(* PLC project PLC, Beckhoff Automation GmbH TwinCAT PLC Control 3.5.13.21 *)
(* stored: creationDateTime 2023-01-03T15:24:25.9685047, modificationDateTime 2023-01-03T15:24:25.9685047 *)

PROGRAM AutoGenerated
  VAR
    Step : INT;
    StepReadEtherCATDiagnostics : INT;
    TonReadDiagnostics : TON;
    sError : STRING;
    FB_EcCoESdoWrite1 : FB_EcCoESdoWrite;
    CoEWriteBuffer : DWORD;
    FB_EcMasterFrameStatisticClearTxRxErr : FB_EcMasterFrameStatisticClearTxRxErr;
    FB_EcGetAllSlavePresentStateChanges : FB_EcGetAllSlavePresentStateChanges;
    fbGetAllSlaveStates : FB_EcGetAllSlaveStates;
    fbEcGetConfSlaves : FB_EcGetConfSlaves;
    fbEcGetAllSlaveCrcErrors : FB_EcGetAllSlaveCrcErrors;
    stSlaveStates : ARRAY[0..EtherDeviceCount] OF ST_EcSlaveState;
    stArrEcConfSlaveInfo : ARRAY[0..EtherDeviceCount] OF ST_EcSlaveConfigData;
    dwArrSlaveCrcCount : ARRAY[0..EtherDeviceCount] OF DWORD;
    dwArrSlaveChangeCount : ARRAY[0..EtherDeviceCount] OF DWORD;
    dwArrSlaveChangeCountHistory : ARRAY[0..EtherDeviceCount] OF DWORD;
    bExecuteFB_GetAdaptersInfo : BOOL := TRUE;  (* /////// Set IP address////////////// *)
    NICCount : INT := 2;
    NicIndex : INT := 1;
    FB_GetAdaptersInfo : FB_GetAdaptersInfo;
    fbDiagRegister : FB_IPCDiag_Register := (sNetId := '');
    fbWriteNicInfo : FB_IPCDiag_WriteParameter;
    iPrevState : INT;
    iState : INT;
    _usiModuleIndex : USINT;
    _sIPAddress : STRING;
    _sIPSubNetMask : STRING;
    _sIPGateway : STRING;
    _xDHCP : BOOL;
    rtExecuteTrig : R_TRIG;
    xBusy : BOOL;
    xError : BOOL;
    hrErrorCode : HRESULT;
    xExecute : BOOL;
    usiModuleIndex : USINT;
    sIPAddress : STRING;
    sIPSubnetMask : STRING;
    sIPGateway : STRING;
    xDHCP : BOOL;
    sCurrentNicName : STRING;
    FB_EcMasterFrameStatisticClearFrames : FB_EcMasterFrameStatisticClearFrames;
    StepCoERead : UDINT;  (* //// End IP address // Start CoE read *)
    CoEReadPos : INT;
    CoEReadbytePos : INT;
    CoEReadintPos : INT;
    CoEReaduintPos : INT;
    CoEReadudintPos : INT;
    CoEReadboolPos : INT;
    fbCoERead : FB_EcCoESdoReadEx;
    CoEReadcbBufLen : ARRAY[1..CoEReadTotalCount] OF UDINT;  (* CoEReadIndex : ARRAY[1..50] OF WORD; CoEReadSubIndex : ARRAY[1..50] OF BYTE; CoEReadSlaveAddr : ARRAY[1..50] OF UINT; *)
    CoEReadData : ARRAY[1..CoEReadTotalCount] OF POINTER TO BYTE;
    CoEReadErrorCounter : UDINT;
    CoEReadErrorIndex : UDINT;
    CoEReadTonUpdateRate : TON;
    i : UDINT;
  END_VAR

            EtherCAT_Diagnostics();

SetIpAddress();
stArrEcConfSlaveInfo[1].sName;
stArrEcConfSlaveInfo[1].sType;
stArrEcConfSlaveInfo[1].nAddr;

CASE StepCoERead OF //Cyclicly read CoE data to send back to rockwell controller.
	0: //This step is important because it sets all the pointer values. 
	
		CoEReadintPos:=0;
		//Not implimented yet.
		CoEReadPos:=1;
		StepCoERead:=StepCoERead+10;
		//Update Pointers
		FOR i:=1 TO  CoEReadTotalCount BY 1 DO
			IF CoEReadDataType[i] = 'INT' THEN
				CoEReadintPos:=CoEReadintPos+1;
				CoEReadData[i]:=ADR(CoEReadInt[CoEReadintPos]);
				CoEReadcbBufLen[i]:=SIZEOF(CoEReadInt[CoEReadintPos]);
			ELSIF CoEReadDataType[i] = 'BYTE' THEN
				CoEReadbytePos:=CoEReadbytePos+1;
				CoEReadData[i]:=ADR(CoEReadByte[CoEReadbytePos]);
				CoEReadcbBufLen[i]:=SIZEOF(CoEReadByte[CoEReadbytePos]);
			ELSIF CoEReadDataType[i] = 'UINT' THEN
				CoEReaduintPos:=CoEReaduintPos+1;
				CoEReadData[i]:=ADR(CoEReadUint[CoEReaduintPos]);
				CoEReadcbBufLen[i]:=SIZEOF(CoEReadUint[CoEReaduintPos]);
			ELSIF CoEReadDataType[i] = 'UDINT' THEN
				CoEReadudintPos:=CoEReadudintPos+1;
				CoEReadData[i]:=ADR(CoEReadUdint[CoEReadudintPos]);
				CoEReadcbBufLen[i]:=SIZEOF(CoEReadUdint[CoEReadudintPos]);
			ELSIF CoEReadDataType[i] = 'BOOL' THEN
				CoEReadboolPos:=CoEReadboolPos+1;
				CoEReadData[i]:=ADR(CoEReadBool[CoEReadboolPos]);
				CoEReadcbBufLen[i]:=SIZEOF(CoEReadBool[CoEReadboolPos]);
			END_IF		
		END_FOR
		
		
	5: //Pause cycle so CoE reads are not constantly occuring.
		CoEReadTonUpdateRate(IN:=TRUE, PT:=T#100MS);	
		IF CoEReadTonUpdateRate.Q THEN
			StepCoERead:=10;
		END_IF
	
	10: //Increment index pointer for next read target.
		fbCoERead( bExecute:=FALSE);
		IF fbCoERead.bBusy = FALSE THEN
			IF CoEReadPos > CoEReadTotalCount THEN
				CoEReadPos:=1;	
				StepCoERead:=5;
				CoEReadTonUpdateRate(IN:=FALSE);		
			ELSE
				IF STRING_TO_UINT(CoEReadSlaveAddress[CoEReadPos]) > 0 AND CoEReadSubIndex[CoEReadPos] > 0  THEN
					//We have something to read		
					StepCoERead:=StepCoERead+10;			
				ELSE
					CoEReadPos:=1;	
					StepCoERead:=5;
					CoEReadTonUpdateRate(IN:=FALSE);		
				END_IF
				
			END_IF
		END_IF
		
	20: //Start read
	fbCoERead(
		sNetId:=F_CreateAmsNetId(nIds := GVL_AutoGenerated.EtherCAT_NetId) , 
		nSlaveAddr:=STRING_TO_UINT(CoEReadSlaveAddress[CoEReadPos]) , 
		nSubIndex:=CoEReadSubIndex[CoEReadPos] , 
		nIndex:=CoEReadIndex[CoEReadPos] , 
		pDstBuf:=CoEReadData[CoEReadPos] , 
		cbBufLen:=CoEReadcbBufLen[CoEReadPos] , 
		bExecute:=TRUE , 
		tTimeout:= , 
		bCompleteAccess:= , 
		bBusy=> , 
		bError=> , 
		nErrId=> , 
		cbRead=> );
	IF NOT fbCoERead.bBusy THEN
		IF fbCoERead.bError THEN
			CoEReadErrorCounter:=CoEReadErrorCounter+1;
			CoEReadErrorIndex:=CoEReadPos;
		END_IF
		CoEReadPos:=CoEReadPos+1;
		StepCoERead:=StepCoERead-10;
	END_IF
END_CASE


CASE Step OF
	0:
		//Not implimented yet.
	
	100:
		IF GVL_AutoGenerated.EtherCAT_CoEWriteExecute THEN
			Step:=Step+10;
		END_IF

		
	110:
	FB_EcCoESdoWrite1(
		sNetId:= , 
		nSlaveAddr:= , 
		nSubIndex:= , 
		nIndex:= , 
		pSrcBuf:= , 
		cbBufLen:= , 
		bExecute:= , 
		tTimeout:= , 
		bBusy=> , 
		bError=> , 
		nErrId=> );
		
	120:
		GVL_AutoGenerated.EtherCAT_CoEWriteDone:=TRUE;
END_CASE


          

METHOD EtherCAT_Diagnostics : BOOL
  VAR
    x : DINT;
  END_VAR
                  
IF EtherCATChangeCountReset THEN
		FOR x :=0 TO EtherDeviceCount BY 1 DO
		dwArrSlaveChangeCountHistory[x]:=dwArrSlaveChangeCount[x];
	END_FOR
END_IF


CASE StepReadEtherCATDiagnostics OF
0:
	FB_EcGetAllSlavePresentStateChanges.bExecute:=FALSE;
	fbGetAllSlaveStates.bExecute:=FALSE;
	fbEcGetConfSlaves.bExecute:=FALSE;
	//fbEcGetAllSlaveCrcErrors.bError:=FALSE;
	TonReadDiagnostics(IN:=TRUE, PT:=T#1S);
	IF TonReadDiagnostics.q THEN
		TonReadDiagnostics(IN:=FALSE);
		StepReadEtherCATDiagnostics:=StepReadEtherCATDiagnostics+10;
		FB_EcGetAllSlavePresentStateChanges.bExecute:=TRUE;
		fbGetAllSlaveStates.bExecute:=TRUE;
		fbEcGetConfSlaves.bExecute:=TRUE;
		//fbEcGetAllSlaveCrcErrors.bError:=TRUE;
	END_IF

10:
	IF NOT FB_EcGetAllSlavePresentStateChanges.bBusy THEN
		StepReadEtherCATDiagnostics:=StepReadEtherCATDiagnostics+10;
		IF NOT FB_EcGetAllSlavePresentStateChanges.bError THEN		
			;
		ELSE
			sError:='fbEcGetAllSlaveAbnormalStateChanges';
		END_IF
	END_IF
	
20:
	IF NOT fbGetAllSlaveStates.bBusy THEN
		StepReadEtherCATDiagnostics:=StepReadEtherCATDiagnostics+10;
		IF fbGetAllSlaveStates.bError THEN
			sError:='fbGetAllSlaveStates';
		END_IF
	END_IF
	
30:
	IF NOT fbEcGetConfSlaves.bBusy THEN
		StepReadEtherCATDiagnostics:=StepReadEtherCATDiagnostics+10;
		IF fbEcGetConfSlaves.bError THEN
			sError:='fbEcGetConfSlaves';
		END_IF
	END_IF
	
40:
	IF NOT fbEcGetAllSlaveCrcErrors.bBusy THEN
		StepReadEtherCATDiagnostics:=StepReadEtherCATDiagnostics+10;
		IF fbEcGetAllSlaveCrcErrors.bError THEN			
			sError:='fbEcGetAllSlaveCrcErrors';
		END_IF
	END_IF
	
50:	//Use this step to copy all the values to PDO to be sent to the EIP network
	StepReadEtherCATDiagnostics:=0;
	FOR x :=0 TO EtherDeviceCount-1 BY 1 DO
	GVL_AutoGenerated.EtherCATChangeCount[x+1]:=DWORD_TO_UINT(dwArrSlaveChangeCount[x] - dwArrSlaveChangeCountHistory[x]);
	GVL_AutoGenerated.EtherCATState[x+1]:=DWORD_TO_UINT(stSlaveStates[x].deviceState);
	END_FOR
END_CASE


FB_EcCoESdoWrite1(
	sNetId:= F_CreateAmsNetId(nIds := GVL_AutoGenerated.EtherCAT_NetId) , 
	nSlaveAddr:=GVL_AutoGenerated.EtherCAT_CoEWriteSlaveAddr , 
	nSubIndex:=GVL_AutoGenerated.EtherCAT_CoEWriteSubIndex , 
	nIndex:= GVL_AutoGenerated.EtherCAT_CoEWriteIndex, 
	pSrcBuf:=ADR(CoEWriteBuffer) , 
	cbBufLen:=SIZEOF(CoEWriteBuffer) , 
	bBusy=> , 
	bError=>GVL_AutoGenerated.EtherCAT_CoEWriteError , 
	nErrId=> );

	
FB_EcGetAllSlavePresentStateChanges(
	sNetId:= F_CreateAmsNetId(nIds := GVL_AutoGenerated.EtherCAT_NetId), 
	pAddrBuf:= ADR(dwArrSlaveChangeCount), 
	cbBufLen:= SIZEOF(dwArrSlaveChangeCount), 
	bExecute:= , 
	tTimeout:= , 
	bBusy=> , 
	bError=> , 
	nErrId=> , 
	nSlaves=> );

fbGetAllSlaveStates(
	sNetId		:=  F_CreateAmsNetId(nIds := GVL_AutoGenerated.EtherCAT_NetId),
	pStateBuf	:= ADR(stSlaveStates),
	cbBufLen	:= SIZEOF(stSlaveStates),
	//bExecute	:=TRUE ,
	tTimeout	:= T#2s);

//fbEcGetConfSlaves(bExecute:=FALSE);
fbEcGetConfSlaves(
	sNetId:=F_CreateAmsNetId(nIds := GVL_AutoGenerated.EtherCAT_NetId),
	pArrEcConfSlaveInfo:=ADR(stArrEcConfSlaveInfo) ,
	cbBufLen:=SIZEOF(stArrEcConfSlaveInfo) ,
	//bExecute:=TRUE ,
	tTimeout:=T#2s  );

//fbEcGetAllSlaveCrcErrors(bExecute:=FALSE);
fbEcGetAllSlaveCrcErrors(
	sNetId:=F_CreateAmsNetId(nIds := GVL_AutoGenerated.EtherCAT_NetId) ,
	pCrcErrorBuf:=ADR(dwArrSlaveCrcCount) ,
	cbBufLen:=SIZEOF(dwArrSlaveCrcCount) ,
	//bExecute:=TRUE 
);
	
                
END_METHOD

METHOD SetIpAddress : BOOL
                  rtExecuteTrig(clk:= xExecute);
usiModuleIndex;
//sIPAddress:=GVL_Constants_AutoGenerated.PLCIPAddress;
//sIPSubnetMask:='255.255.255.0';
//xDHCP:=false;
//sIPAddress := PLCIPAddress001;

FB_GetAdaptersInfo.arrAdapters[0].bDhcpEnabled;
FB_GetAdaptersInfo.arrAdapters[1].bDhcpEnabled;
FB_GetAdaptersInfo.arrAdapters[0].sIpAddr;
FB_GetAdaptersInfo.arrAdapters[1].sIpAddr;
FB_GetAdaptersInfo.arrAdapters[1].physAddr;



FB_GetAdaptersInfo(
	sNetID:= , 
	bExecute:=bExecuteFB_GetAdaptersInfo , 
	tTimeout:= , 
	bBusy=> , 
	bError=> , 
	nErrID=> , 
	arrAdapters=> , 
	nCount=> , 
	nGet=> );

CASE iState OF
	0:	// Init
		IF NOT fbDiagRegister.bBusy THEN
			fbDiagRegister(bExecute:=TRUE); // need to be executed once
		ELSE
			fbDiagRegister(bExecute:=FALSE);
		END_IF
		IF NOT fbDiagRegister.bBusy AND NOT FB_GetAdaptersInfo.bBusy THEN
			iPrevState:= iState;
			iState := SEL(fbDiagRegister.bError, 1, 99);
			bExecuteFB_GetAdaptersInfo:=FALSE;
		END_IF
		
	1:	// Wait for execute
		IF NicIndex <= NICCount THEN
			iPrevState:= iState;
			iState:= iState+1;
			usiModuleIndex := INT_TO_USINT(NicIndex);
			sCurrentNicName := FB_GetAdaptersInfo.arrAdapters[NicIndex-1].sDescription;
			IF NicIndex = 1 THEN		
				//usiModuleIndex:=1;
				IF PLCIPAddress001 = 'DHCP' THEN
					xDHCP:=TRUE;
				ELSE
					sIPSubnetMask:='255.255.255.0';
					xDHCP:=FALSE;
					sIPAddress := PLCIPAddress001;
				END_IF
			END_IF
			IF NicIndex = 2 THEN
				//usiModuleIndex:=0;
				IF PLCIPAddress000 = 'DHCP' THEN
					xDHCP:=TRUE;
				ELSE
					sIPSubnetMask:='255.255.255.0';
					xDHCP:=FALSE;
					sIPAddress := PLCIPAddress000;
				END_IF		
			END_IF
		END_IF
	
	2:
	
		fbWriteNicInfo(bExecute:= FALSE, fbRegister:= fbDiagRegister);
		hrErrorCode:= 0;
		xBusy:= TRUE;
		xError:= FALSE;
		IF usiModuleIndex > 0 
			AND (xDHCP OR (sIPAddress <> '' AND sIPSubnetMask <> '')) THEN
				_usiModuleIndex:= usiModuleIndex;
				_sIPAddress:= sIPAddress;
				_sIPSubNetMask:= sIPSubnetMask;
				_sIPGateway:= sIPGateway;
				_xDHCP:= xDHCP;
				iPrevState:= iState;
				iState:= 20;					
		ELSE
			iPrevState:= iState;
			iState:= 99;	
		END_IF				


		
	20:	// Write DHCP
		fbWriteNicInfo(
			bExecute:= TRUE, 
			eParameterKey:= E_IPCDiag_ParameterKey.NIC_DHCP, 
			pBuffer:= ADR(_xDHCP), 
			nBufferSize:= SIZEOF(_xDHCP), 
			nModuleIdx:= _usiModuleIndex, 
			nListIdx:= , 
			tTimeout:= T#5S, 
			sNetId:= '', 
			xReserved:= , 
			fbRegister:= fbDiagRegister, 
			bBusy=> , 
			bError=> , 
			hrErrorCode=> , 
			ipErrorMessage=> );
	
		IF NOT fbWriteNicInfo.bBusy THEN
			IF NOT fbWriteNicInfo.bError THEN
				fbWriteNicInfo(bExecute:= FALSE, fbRegister:= fbDiagRegister);
				iPrevState:= iState;
				iState:= iState + 10;
				IF _xDHCP THEN
					iState:= 60;
				END_IF
			ELSE
				iPrevState:= iState;
				iState:= 99;
			END_IF
		END_IF
		
	30: // Write IP Address
		fbWriteNicInfo(
			bExecute:= TRUE, 
			eParameterKey:= E_IPCDiag_ParameterKey.NIC_IPv4Address, 
			pBuffer:= ADR(_sIPAddress), 
			nBufferSize:= SIZEOF(_sIPAddress), 
			nModuleIdx:= _usiModuleIndex, 
			nListIdx:= , 
			tTimeout:= T#5S, 
			sNetId:= '', 
			xReserved:= , 
			fbRegister:= fbDiagRegister, 
			bBusy=> , 
			bError=> , 
			hrErrorCode=> , 
			ipErrorMessage=> );
	
		IF NOT fbWriteNicInfo.bBusy THEN
			IF NOT fbWriteNicInfo.bError THEN
				fbWriteNicInfo(bExecute:= FALSE, fbRegister:= fbDiagRegister);
				iPrevState:= iState;
				iState:= iState + 10;
			ELSE
				iPrevState:= iState;
				iState:= 99;
			END_IF
		END_IF	
	
	40:	// Write Subnet Mask
		fbWriteNicInfo(
			bExecute:= TRUE, 
			eParameterKey:= E_IPCDiag_ParameterKey.NIC_IPv4SubnetMask, 
			pBuffer:= ADR(_sIPSubNetMask), 
			nBufferSize:= SIZEOF(_sIPSubNetMask), 
			nModuleIdx:= _usiModuleIndex, 
			nListIdx:= , 
			tTimeout:= T#5S, 
			sNetId:= '', 
			xReserved:= , 
			fbRegister:= fbDiagRegister, 
			bBusy=> , 
			bError=> , 
			hrErrorCode=> , 
			ipErrorMessage=> );
	
		IF NOT fbWriteNicInfo.bBusy THEN
			IF NOT fbWriteNicInfo.bError THEN
				fbWriteNicInfo(bExecute:= FALSE, fbRegister:= fbDiagRegister);
				iPrevState:= iState;
				iState:= iState + 10;
			ELSE
				iPrevState:= iState;
				iState:= 99;
			END_IF
		END_IF		
	
	50:	// Write Gateway
		fbWriteNicInfo(
			bExecute:= TRUE, 
			eParameterKey:= E_IPCDiag_ParameterKey.NIC_IPv4DefGateway, 
			pBuffer:= ADR(_sIPGateway), 
			nBufferSize:= SIZEOF(_sIPGateway), 
			nModuleIdx:= _usiModuleIndex, 
			nListIdx:= , 
			tTimeout:= T#5S, 
			sNetId:= '', 
			xReserved:= , 
			fbRegister:= fbDiagRegister, 
			bBusy=> , 
			bError=> , 
			hrErrorCode=> , 
			ipErrorMessage=> );
	
		IF NOT fbWriteNicInfo.bBusy THEN
			IF NOT fbWriteNicInfo.bError THEN
				fbWriteNicInfo(bExecute:= FALSE, fbRegister:= fbDiagRegister);
				iPrevState:= iState;
				iState:= iState + 10;
			ELSE
				iPrevState:= iState;
				iState:= 99;
			END_IF
		END_IF		
		
	60:
		xBusy:= FALSE;
		xError:= FALSE;
		iPrevState:= iState;
		iState:= 0;
		NicIndex:=NicIndex+1;
		bExecuteFB_GetAdaptersInfo:=TRUE;
	
	99:
		xBusy:= FALSE;
		xError:= TRUE;
		hrErrorCode:= fbWriteNicInfo.hrErrorCode;
		IF NOT xExecute THEN
			iPrevState:= iState;
			iState:= 0;
		END_IF
	
END_CASE

                
END_METHOD
END_PROGRAM
